(* PLC project actuator, TNI-Software ControlBuild 4.00.17 *)
(* stored: creationDateTime 2005-06-20T11:52:29-01:00 *)

FUNCTION_BLOCK cmd_equipment_library.actuator
  VAR_INPUT  (* CB.group=Modes CB.kind=inputVars *)
    autoMode : BOOL := false;  (* CB.libelle=Automatic mode *)
    manualMode : BOOL := false;  (* CB.libelle=Manual mode *)
  END_VAR
  VAR_INPUT  (* CB.group=Commands CB.kind=inputVars *)
    autoCmd : BOOL := false;  (* CB.libelle=Automatic command *)
  END_VAR
  VAR_INPUT  (* CB.group=PushButtons CB.kind=inputVars *)
    forwardPB : BOOL := false;  (* CB.libelle=Forward pushbutton *)
    stopPB : BOOL := false;  (* CB.libelle=Stop pushbutton *)
  END_VAR
  VAR_INPUT  (* CB.kind=inputVars *)
    generalFault : BOOL := false;  (* CB.mnemonicPatternPropertyName=<SY>_DEF_<NU> CB.libelle=General fault of the engine *)
  END_VAR
  VAR_OUTPUT  (* CB.group=Orders CB.kind=outputVars *)
    forwardCmd : BOOL := false;  (* CB.mnemonicPatternPropertyName=fwdCmd<SY><NU> CB.libelle=Forward command *)
  END_VAR

(* LD diagram, written out as Structured Text *)
1:
forwardCmd := (autoMode AND autoCmd OR manualMode AND (forwardPB OR forwardCmd) AND NOT stopPB) AND NOT generalFault;
END_FUNCTION_BLOCK
